// TwinCAT 3 PLC project Untitled1
// ProgramVersion: 3.1.4024.0
// libraries:
//   SPT Base Types, * (Beckhoff Automation LLC)
//   SPT Components, * (Beckhoff Automation LLC)
//   SPT Event Logger, * (Beckhoff Automation LLC)
//   SPT Motion Control, * (Beckhoff Automation LLC)
//   Tc2_EtherCAT, * (Beckhoff Automation GmbH)
//   Tc2_Standard, * (Beckhoff Automation GmbH)
//   Tc2_System, * (Beckhoff Automation GmbH)
//   Tc3_EventLogger, * (Beckhoff Automation GmbH)
//   Tc3_Module, * (Beckhoff Automation GmbH)
//   Tc3_PackML_V2, * (Beckhoff Automation GmbH)
// project tree:
//   DUTs/ E_PMLCustomMode.TcDUT
//   Machine/01_MachineModule/DUTs/ ST_MachineCommand.TcDUT, ST_MachineConfig.TcDUT, ST_MachineRecipe.TcDUT, ST_MachineStatus.TcDUT
//   Machine/01_MachineModule/ I_MachineModule.TcIO, Machine.TcPOU
//   Machine/02_EquipmentModules/01_Infeed/DUTs/ ST_InfeedConfig.TcDUT, ST_InfeedRecipe.TcDUT, ST_InfeedStatus.TcDUT, ST_InfeedCommand.TcDUT
//   Machine/02_EquipmentModules/01_Infeed/ EM_InfeedModule.TcPOU, I_InfeedModule.TcIO
//   Machine/02_EquipmentModules/02_Process/DUTs/ ST_ProcessCommand.TcDUT, ST_ProcessConfig.TcDUT, ST_ProcessRecipe.TcDUT, ST_ProcessStatus.TcDUT
//   Machine/02_EquipmentModules/02_Process/ EM_ProcessModule.TcPOU, I_ProcessModule.TcIO
//   Machine/02_EquipmentModules/03_Outfeed/DUTs/ ST_OutfeedCommand.TcDUT, ST_OutfeedConfig.TcDUT, ST_OutfeedRecipe.TcDUT, ST_OutfeedStatus.TcDUT
//   Machine/02_EquipmentModules/03_Outfeed/ EM_OutfeedModule.TcPOU, I_OutfeedModule.TcIO
//   Machine/03_Components/ FB_Component_StackLight.TcPOU, FB_Component_TwinSAFE_Monitor.TcPOU
//   / PlcTask.TcTTO
//   POUs/ CD_CommonModule.TcCD (not stored), CD_Visitor.TcCD (not stored), MAIN.TcPOU
//   POUs/Common/Component/ CommonComponent.TcPOU, I_CommonComponent.TcIO
//   POUs/Common/Module/ CommonModule.TcPOU, I_CommonModule.TcIO
//   POUs/Common/Module/DUTs/ ST_CommandCommon.TcDUT, ST_ConfigCommon.TcDUT, ST_RecipeCommon.TcDUT, ST_StatusCommon.TcDUT
//   Visitors/ FB_CollectOEE.TcPOU, I_VisitModules.TcIO
// real-time tasks:
//   TASK PlcTask: cycle T#10ms, priority 20, ADS port 350
// motion (NC):
//   TASK NC-Task 1 SAF: cycle T#2ms, priority 4, ADS port 501
//   TASK NC-Task 1 SVB: cycle T#10ms, priority 8, ADS port 511
//   AXIS Infeed (id 1)
//     OtherSettings: AllowMotionCmdToSlave=true
//     encoder EncType=1
//     drive DrvType=5
//       Analog: TorqueSetpointScale=10, ScaleFactorActTorque=0.1
//     controller CtrType=1
//       CtrPara: PriorControlFactor=1
//         Observer: BandWidth=20
//   AXIS Process (id 2)
//     OtherSettings: AllowMotionCmdToSlave=true
//     encoder EncType=1
//     drive DrvType=5
//       Analog: TorqueSetpointScale=10, ScaleFactorActTorque=0.1
//     controller CtrType=1
//       CtrPara: PriorControlFactor=1
//         Observer: BandWidth=20
//   AXIS Outfeed (id 3)
//     OtherSettings: AllowMotionCmdToSlave=true
//     encoder EncType=1
//     drive DrvType=5
//       Analog: TorqueSetpointScale=10, ScaleFactorActTorque=0.1
//     controller CtrType=1
//       CtrPara: PriorControlFactor=1
//         Observer: BandWidth=20
// variable links:
//   Untitled1/Untitled1 Instance <-> NC-Task 1 SAF/Axes/Infeed
//     PlcTask Inputs/MAIN.Machine.Infeed.Axis.BasicAxis._Axis.NcToPlc <-> Outputs/ToPlc
//     PlcTask Outputs/MAIN.Machine.Infeed.Axis.BasicAxis._Axis.PlcToNc <-> Inputs/FromPlc
//   Untitled1/Untitled1 Instance <-> NC-Task 1 SAF/Axes/Outfeed
//     PlcTask Inputs/MAIN.Machine.Outfeed.Axis.BasicAxis._Axis.NcToPlc <-> Outputs/ToPlc
//     PlcTask Outputs/MAIN.Machine.Outfeed.Axis.BasicAxis._Axis.PlcToNc <-> Inputs/FromPlc
//   Untitled1/Untitled1 Instance <-> NC-Task 1 SAF/Axes/Process
//     PlcTask Inputs/MAIN.Machine.Process.Axis.BasicAxis._Axis.NcToPlc <-> Outputs/ToPlc
//     PlcTask Outputs/MAIN.Machine.Process.Axis.BasicAxis._Axis.PlcToNc <-> Inputs/FromPlc

CONFIGURATION Untitled1
    RESOURCE PLC ON TwinCAT3
        TASK PlcTask(INTERVAL := T#10ms, PRIORITY := 20);
        PROGRAM MAIN WITH PlcTask : MAIN;
    END_RESOURCE
END_CONFIGURATION

// ---- DUTs/E_PMLCustomMode.TcDUT
{attribute 'to_string'}
TYPE E_PMLCustomMode : (
		//Reserved
		Production	:= 1,
		Maintenance := 2,
		Manual		:= 3,
		//User-Defined
		Home		   := 4,
		PrePositioning := 5,
		PreHeating	   := 6,
		PreProduction  := 7,
		SingleCycle	   := 8,
		SingleStep	   := 9,
		SetupMode	   := 10,
		CleanInPlace   := 11
	) DINT;
END_TYPE

// ---- Machine/01_MachineModule/DUTs/ST_MachineCommand.TcDUT
TYPE ST_MachineCommand :
	STRUCT
		LightOn : BOOL;
	END_STRUCT
END_TYPE

// ---- Machine/01_MachineModule/DUTs/ST_MachineConfig.TcDUT
TYPE ST_MachineConfig :
	STRUCT
	END_STRUCT
END_TYPE

// ---- Machine/01_MachineModule/DUTs/ST_MachineRecipe.TcDUT
TYPE ST_MachineRecipe :
	STRUCT
	END_STRUCT
END_TYPE

// ---- Machine/01_MachineModule/DUTs/ST_MachineStatus.TcDUT
TYPE ST_MachineStatus :
	STRUCT
	END_STRUCT
END_TYPE

// ---- Machine/02_EquipmentModules/01_Infeed/DUTs/ST_InfeedConfig.TcDUT
TYPE ST_InfeedConfig :
	STRUCT
	END_STRUCT
END_TYPE

// ---- Machine/02_EquipmentModules/01_Infeed/DUTs/ST_InfeedRecipe.TcDUT
TYPE ST_InfeedRecipe :
	STRUCT
	END_STRUCT
END_TYPE

// ---- Machine/02_EquipmentModules/01_Infeed/DUTs/ST_InfeedStatus.TcDUT
TYPE ST_InfeedStatus :
	STRUCT
		ConveyorRunning : BOOL;
	END_STRUCT
END_TYPE

// ---- Machine/02_EquipmentModules/01_Infeed/DUTs/ST_InfeedCommand.TcDUT
TYPE ST_InfeedCommand :
	STRUCT
		StartConveyor : BOOL;
		StopConveyor  : BOOL;
	END_STRUCT
END_TYPE

// ---- Machine/02_EquipmentModules/02_Process/DUTs/ST_ProcessCommand.TcDUT
TYPE ST_ProcessCommand :
	STRUCT
		MoveToAbortPos : BOOL;
	END_STRUCT
END_TYPE

// ---- Machine/02_EquipmentModules/02_Process/DUTs/ST_ProcessConfig.TcDUT
TYPE ST_ProcessConfig :
	STRUCT
	END_STRUCT
END_TYPE

// ---- Machine/02_EquipmentModules/02_Process/DUTs/ST_ProcessRecipe.TcDUT
TYPE ST_ProcessRecipe :
	STRUCT
		RollTime : TIME := T#1S;
	END_STRUCT
END_TYPE

// ---- Machine/02_EquipmentModules/02_Process/DUTs/ST_ProcessStatus.TcDUT
TYPE ST_ProcessStatus :
	STRUCT
		ProductAtReady	: BOOL;
		ProductInPos	: BOOL;
		ProcessComplete : BOOL;
	END_STRUCT
END_TYPE

// ---- Machine/02_EquipmentModules/03_Outfeed/DUTs/ST_OutfeedCommand.TcDUT
TYPE ST_OutfeedCommand :
	STRUCT
		StartConveyor : bool;
		StopConveyor : BOOL;
	END_STRUCT
END_TYPE

// ---- Machine/02_EquipmentModules/03_Outfeed/DUTs/ST_OutfeedConfig.TcDUT
TYPE ST_OutfeedConfig :
	STRUCT
	END_STRUCT
END_TYPE

// ---- Machine/02_EquipmentModules/03_Outfeed/DUTs/ST_OutfeedRecipe.TcDUT
TYPE ST_OutfeedRecipe :
	STRUCT
	END_STRUCT
END_TYPE

// ---- Machine/02_EquipmentModules/03_Outfeed/DUTs/ST_OutfeedStatus.TcDUT
TYPE ST_OutfeedStatus :
	STRUCT
		ProductAtReady	: BOOL;
		ProductRemoved	: BOOL;
		ConveyorRunning : BOOL;
	END_STRUCT
END_TYPE

// ---- POUs/Common/Module/DUTs/ST_CommandCommon.TcDUT
TYPE ST_CommandCommon EXTENDS ST_PackMLBaseModule_Command :
	STRUCT
		Home		   : BOOL;
		Start		   : BOOL;
		Reset		   : BOOL;
		EmergencyStop  : BOOL;
		ControlledStop : BOOL;
	END_STRUCT
END_TYPE

// ---- POUs/Common/Module/DUTs/ST_ConfigCommon.TcDUT
TYPE ST_ConfigCommon :
STRUCT
END_STRUCT
END_TYPE

// ---- POUs/Common/Module/DUTs/ST_RecipeCommon.TcDUT
TYPE ST_RecipeCommon :
STRUCT
END_STRUCT
END_TYPE

// ---- POUs/Common/Module/DUTs/ST_StatusCommon.TcDUT
TYPE ST_StatusCommon EXTENDS ST_PackMLBaseModule_Status :
	STRUCT
		Homed : BOOL;
	END_STRUCT
END_TYPE

// ---- Machine/01_MachineModule/I_MachineModule.TcIO
INTERFACE I_MachineModule

PROPERTY CfgMachine : REFERENCE TO ST_MachineConfig
GET
END_GET
END_PROPERTY

PROPERTY CmdMachine : REFERENCE TO ST_MachineCommand
GET
END_GET
END_PROPERTY

PROPERTY RcpMachine : REFERENCE TO ST_MachineRecipe
GET
END_GET
END_PROPERTY

PROPERTY StsMachine : REFERENCE TO ST_MachineStatus
GET
END_GET
END_PROPERTY

END_INTERFACE

// ---- Machine/02_EquipmentModules/01_Infeed/I_InfeedModule.TcIO
INTERFACE I_InfeedModule

PROPERTY CfgInfeed : REFERENCE TO ST_InfeedConfig
GET
END_GET
END_PROPERTY

PROPERTY CmdInfeed : REFERENCE TO ST_InfeedCommand
GET
END_GET
END_PROPERTY

PROPERTY RcpInfeed : REFERENCE TO ST_InfeedRecipe
GET
END_GET
END_PROPERTY

PROPERTY StsInfeed : REFERENCE TO ST_InfeedStatus
GET
END_GET
END_PROPERTY

END_INTERFACE

// ---- Machine/02_EquipmentModules/02_Process/I_ProcessModule.TcIO
INTERFACE I_ProcessModule

PROPERTY CfgProcess : REFERENCE TO ST_ProcessConfig
GET
END_GET
END_PROPERTY

PROPERTY CmdProcess : REFERENCE TO ST_ProcessCommand
GET
END_GET
END_PROPERTY

PROPERTY RcpProcess : REFERENCE TO ST_ProcessRecipe
GET
END_GET
END_PROPERTY

PROPERTY StsProcess : REFERENCE TO ST_ProcessStatus
GET
END_GET
END_PROPERTY

END_INTERFACE

// ---- Machine/02_EquipmentModules/03_Outfeed/I_OutfeedModule.TcIO
INTERFACE I_OutfeedModule

PROPERTY CfgOutfeed : REFERENCE TO ST_OutfeedConfig
GET
END_GET
END_PROPERTY

PROPERTY CmdOutfeed : REFERENCE TO ST_OutfeedCommand
GET
END_GET
END_PROPERTY

PROPERTY RcpOutfeed : REFERENCE TO ST_OutfeedRecipe
GET
END_GET
END_PROPERTY

PROPERTY StsOutfeed : REFERENCE TO ST_OutfeedStatus
GET
END_GET
END_PROPERTY

END_INTERFACE

// ---- POUs/Common/Component/I_CommonComponent.TcIO
INTERFACE I_CommonComponent EXTENDS I_ComponentBase

END_INTERFACE

// ---- POUs/Common/Module/I_CommonModule.TcIO
INTERFACE I_CommonModule EXTENDS I_PackML_BaseModule

METHOD Accept
VAR_INPUT
	Visitor : I_VisitModules;
END_VAR
END_METHOD

PROPERTY CfgCommon : reference to ST_ConfigCommon
GET
END_GET
END_PROPERTY

PROPERTY CmdCommon : REFERENCE TO ST_CommandCommon
GET
END_GET
END_PROPERTY

PROPERTY RcpCommon : reference to ST_RecipeCommon
GET
END_GET
END_PROPERTY

PROPERTY StsCommon : REFERENCE TO ST_StatusCommon
GET
END_GET
END_PROPERTY

END_INTERFACE

// ---- Visitors/I_VisitModules.TcIO
INTERFACE I_VisitModules

METHOD VisitModule : BOOL
VAR_INPUT
	Module : I_CommonModule;
END_VAR
END_METHOD

END_INTERFACE

// ---- POUs/MAIN.TcPOU
PROGRAM MAIN
VAR
	Machine		   : Machine := (Name := 'Machine');
	Reset		   : BOOL;
	Home		   : BOOL;
	Start		   : BOOL;
	Stop		   : BOOL;
	ControlledStop : BOOL;
	EmergencyStop  : BOOL;
END_VAR

(*
	This sample was built to show a few different ways of implementing the various parts of the SPT Framework.
	While the SPT Framework provides the FB_PackML_BaseModule, this Class focuses on providing the necessities from which to build upon.
	
	This sample uses a CommonModule Class that inheirts from the FB_PackML_BaseModule, and does most of the work for managing the state machine of the system's modules.
		This allows for the code that interacts with the Components of a Module to be the primary focuis of the EM.
 	The CommonModule implements the Command and Status Structures which allows for interaction with a modules state machine. Common commands such as Start, Stop, Reset, and Home 
		are sent through the CmdCommon structure. Common Status of the modules can be read through the StsCommon structure.
	For consistency each Equipment Module also has a Cmd and Sts structure named for the EM; for example, CmdInfeed or StsProcess. 
		These hold the more specific EM commands such as Conveyor Start and Conveyor Stop, and a similar Status structure for Conveyor Running or Cylinder Extended.
		It is important to note that all of these structures have a concrete instance defined within the EM, and a property getter that gets a reference to that concretion. 
		This means that it is possible to read and write to the structure through the getter of the propoerty.
	This overall design allows for the code to Stop, Reset, Enable/Disable; that most all components are going to need, to be placed in the CommonModule. Thereby providing the possibility
		to reduce the code in the EMs to only managing what is unique about the EM. This does require the use of interfaces and the __QUERYINTERFACE method, 
		in order to only send axis command to an axis, but it does allow us to efficiently send commands to all axes within an EM at the same time.
		Additionally, if components built by the user implement a common interface to a structure then these components can all be managed through that interface from the CommonModule.
		
	IMPORTANT NOTE:
	The CommonModule makes extensive use of the variable SequenceState throughout the Acting and Execute methods. 
	Therefore it is reccomend to only use the DescendantSequenceState variable within the EMs.
	
*)
Machine.CyclicLogic();

(*
If Not Homed Abort -> Idle, Change Mode to Home, Idle -> Execute
If Homed Abort -> Idle in Mode Production *)
IF Reset THEN
	Reset					:= FALSE;
	Machine.CmdCommon.Reset := TRUE; //Needs to be ignored if state not valid for reset
END_IF

(*
In Home.Execute start Homing Sequence
After Homing finished, Execute -> Suspended, ModeChange to Production *)
IF Home THEN
	Home				   := FALSE;
	Machine.CmdCommon.Home := TRUE; ////Needs to be ignored if state not valid for Home
END_IF

(*
Production.Idle -> Execute
Production.Suspended -> Execute *)
IF Start THEN
	Start					:= FALSE;
	Machine.CmdCommon.Start := TRUE; //Needs to be ignored if state not valid for start
END_IF

IF ControlledStop THEN
	ControlledStop					 := FALSE;
	Machine.CmdCommon.ControlledStop := TRUE;
	Machine.ChangeState(State := E_PMLCommand.ePMLCommand_Stop);
END_IF

IF EmergencyStop THEN
	EmergencyStop					:= FALSE;
	Machine.CmdCommon.EmergencyStop := TRUE;
	Machine.ChangeState(State := E_PMLCommand.ePMLCommand_Abort);
END_IF

END_PROGRAM

// ---- Machine/01_MachineModule/Machine.TcPOU
FUNCTION_BLOCK Machine EXTENDS CommonModule IMPLEMENTS I_MachineModule
VAR
	//EMs
	Infeed	: EM_InfeedModule  := (Name := 'Infeed');
	Process : EM_ProcessModule := (Name := 'Process');
	Outfeed : EM_OutfeedModule := (Name := 'Outfeed');

	//Components
	StackLight		 : FB_Component_StackLight		 := (Name := 'StackLight');
	TwinSAFE_Monitor : FB_Component_TwinSAFE_Monitor := (Name := 'TwinSAFE_Monitor');

	//
	fbTON_InfeedRun	   : TON;
	fbTON_ProcessDelay : TON;
	fbTON_OutfeedRun   : TON;

	//
	_CmdMachine : ST_MachineCommand;
	_StsMachine : ST_MachineStatus;
	_RcpMachine : ST_MachineRecipe;
	_CfgMachine : ST_MachineConfig;

	//Visitor
	CollectOEE_MM : FB_CollectOEE;
END_VAR

PROPERTY CfgMachine : REFERENCE TO ST_MachineConfig
GET
CfgMachine REF= _CfgMachine;
END_GET
END_PROPERTY

PROPERTY CmdMachine : REFERENCE TO ST_MachineCommand
GET
CmdMachine REF= _CmdMachine;
END_GET
END_PROPERTY

METHOD CreateCustomModes : BOOL
VAR_INPUT
END_VAR
//Production
CustomModes(eMode						   := E_PMLCustomMode.Production,
			sName						   := 'Production',
			bDisableClearing			   := FALSE,
			bDisableStarting			   := FALSE,
			bDisableSuspended			   := FALSE,
			bDisableStopping			   := FALSE,
			bDisableAborting			   := FALSE,
			bDisableHolding				   := FALSE,
			bDisableHeld				   := FALSE,
			bDisableUnholding			   := FALSE,
			bDisableSuspending			   := FALSE,
			bDisableUnsuspending		   := FALSE,
			bDisableResetting			   := FALSE,
			bDisableIdle				   := FALSE,
			bDisableCompleting			   := FALSE,
			bDisableComplete			   := FALSE,
			bEnableUnitModeChangeStopped   := TRUE,
			bEnableUnitModeChangeIdle	   := TRUE,
			bEnableUnitModeChangeSuspended := TRUE,
			bEnableUnitModeChangeExecute   := TRUE,
			bEnableUnitModeChangeAborted   := TRUE,
			bEnableUnitModeChangeHeld	   := TRUE,
			bEnableUnitModeChangeComplete  := TRUE);

//Home
CustomModes(eMode						   := E_PMLCustomMode.Home,
			sName						   := 'Home',
			bDisableClearing			   := FALSE,
			bDisableStarting			   := FALSE,
			bDisableSuspended			   := FALSE,
			bDisableStopping			   := FALSE,
			bDisableAborting			   := FALSE,
			bDisableHolding				   := FALSE,
			bDisableHeld				   := FALSE,
			bDisableUnholding			   := FALSE,
			bDisableSuspending			   := FALSE,
			bDisableUnsuspending		   := FALSE,
			bDisableResetting			   := FALSE,
			bDisableIdle				   := FALSE,
			bDisableCompleting			   := FALSE,
			bDisableComplete			   := FALSE,
			bEnableUnitModeChangeStopped   := TRUE,
			bEnableUnitModeChangeIdle	   := TRUE,
			bEnableUnitModeChangeSuspended := TRUE,
			bEnableUnitModeChangeExecute   := TRUE,
			bEnableUnitModeChangeAborted   := TRUE,
			bEnableUnitModeChangeHeld	   := TRUE,
			bEnableUnitModeChangeComplete  := TRUE);

//Pre-Positioning for resetting between products
CustomModes(eMode						   := E_PMLCustomMode.PrePositioning,
			sName						   := 'Pre-Positioning',
			bDisableClearing			   := FALSE,
			bDisableStarting			   := FALSE,
			bDisableSuspended			   := FALSE,
			bDisableStopping			   := FALSE,
			bDisableAborting			   := FALSE,
			bDisableHolding				   := FALSE,
			bDisableHeld				   := FALSE,
			bDisableUnholding			   := FALSE,
			bDisableSuspending			   := FALSE,
			bDisableUnsuspending		   := FALSE,
			bDisableResetting			   := FALSE,
			bDisableIdle				   := FALSE,
			bDisableCompleting			   := FALSE,
			bDisableComplete			   := FALSE,
			bEnableUnitModeChangeStopped   := TRUE,
			bEnableUnitModeChangeIdle	   := TRUE,
			bEnableUnitModeChangeSuspended := TRUE,
			bEnableUnitModeChangeExecute   := TRUE,
			bEnableUnitModeChangeAborted   := TRUE,
			bEnableUnitModeChangeHeld	   := TRUE,
			bEnableUnitModeChangeComplete  := TRUE);

//Pre-Production for Heaters
CustomModes(eMode						   := E_PMLCustomMode.PreProduction,
			sName						   := 'Pre-Production',
			bDisableClearing			   := FALSE,
			bDisableStarting			   := FALSE,
			bDisableSuspended			   := FALSE,
			bDisableStopping			   := FALSE,
			bDisableAborting			   := FALSE,
			bDisableHolding				   := FALSE,
			bDisableHeld				   := FALSE,
			bDisableUnholding			   := FALSE,
			bDisableSuspending			   := FALSE,
			bDisableUnsuspending		   := FALSE,
			bDisableResetting			   := FALSE,
			bDisableIdle				   := FALSE,
			bDisableCompleting			   := FALSE,
			bDisableComplete			   := FALSE,
			bEnableUnitModeChangeStopped   := TRUE,
			bEnableUnitModeChangeIdle	   := TRUE,
			bEnableUnitModeChangeSuspended := TRUE,
			bEnableUnitModeChangeExecute   := TRUE,
			bEnableUnitModeChangeAborted   := TRUE,
			bEnableUnitModeChangeHeld	   := TRUE,
			bEnableUnitModeChangeComplete  := TRUE);
END_METHOD

METHOD PUBLIC CyclicLogic
IF NOT _InitComplete THEN
	_InitComplete := Initialize();
	RETURN;
END_IF

//Visitor
Accept(Visitor := CollectOEE_MM);
SUPER^.CyclicLogic();
END_METHOD

//! @summary This method contains code which will execute when this PackML module is in the <b>Execute</b> state
METHOD PROTECTED Execute
(*! <description> <b>The base implementation of this method is empty. User must override this method to provide functionality.</b>
<table> 
	<tr>
		<th> Previous State </th>
		<th> Transition In </th>
		<th> Transition Out </th>
		<th> Next State  </th> 
	</tr>
	<tr>
		<td> Starting<b>-or-</b>Unholding <b>-or-</b>Unsuspending</td>
		<td> State Complete<i>(Starting<b>-or-</b>Unholding<b>-or-</b>Unsuspending)</i></td> 
		<td> State Complete<b>-or-</b>Hold Command<b>-or-</b>Suspend Command</td>
		<td> Completing<b>-or-</b>Holding<b>-or-</b>Suspending</td>
	</tr>
</table>
This method is called as required by <c>StateControl()</c>
</description> 

*)
VAR
END_VAR
CASE _CurrentMode OF
	E_PMLCustomMode.Production:
		CASE DescendantSequenceState OF
			0:
				Infeed.CmdInfeed.StartConveyor := TRUE;
				IF Infeed.StsInfeed.ConveyorRunning THEN
					Infeed.CmdInfeed.StartConveyor := FALSE;
					fbTON_InfeedRun(IN := FALSE);
					DescendantSequenceState := DescendantSequenceState + 10;
				END_IF

			10:
				fbTON_InfeedRun(IN := TRUE, PT := T#3S);
				IF fbTON_InfeedRun.Q THEN
					Infeed.CmdInfeed.StopConveyor := TRUE;
					DescendantSequenceState		  := DescendantSequenceState + 10;
				END_IF

			20:
				IF NOT Infeed.StsInfeed.ConveyorRunning THEN
					Infeed.CmdInfeed.StopConveyor	  := FALSE;
					Process.StsProcess.ProductAtReady := TRUE;
					fbTON_ProcessDelay(IN := FALSE);
					DescendantSequenceState := DescendantSequenceState + 10;
				END_IF

			30:
				fbTON_ProcessDelay(IN := TRUE, PT := T#1.5S);
				IF fbTON_ProcessDelay.Q THEN
					Process.StsProcess.ProductAtReady := FALSE;
					Process.StsProcess.ProductInPos	  := TRUE;
					DescendantSequenceState			  := DescendantSequenceState + 10;
				END_IF

			40:
				IF Process.StsProcess.ProcessComplete THEN
					Process.StsProcess.ProcessComplete := FALSE;
					Outfeed.StsOutfeed.ProductAtReady  := TRUE;
					DescendantSequenceState			   := DescendantSequenceState + 10;
				END_IF

			50:
				IF Outfeed.StsOutfeed.ConveyorRunning THEN
					Outfeed.StsOutfeed.ProductAtReady := FALSE;
					fbTON_OutfeedRun(IN := FALSE);
					DescendantSequenceState := DescendantSequenceState + 10;
				END_IF

			60:
				fbTON_OutfeedRun(IN := TRUE, PT := T#3S);
				IF fbTON_OutfeedRun.Q THEN
					Outfeed.StsOutfeed.ProductRemoved := TRUE;
					DescendantSequenceState			  := DescendantSequenceState + 10;
				END_IF

			70:
				IF NOT Outfeed.StsOutfeed.ConveyorRunning THEN
					Outfeed.StsOutfeed.ProductRemoved := FALSE;
					DescendantSequenceState			  := 0;
				END_IF
		END_CASE

	E_PMLCustomMode.Home:
		_StsCommon.Homed := TRUE;
END_CASE

SUPER^.Execute();
END_METHOD

METHOD PROTECTED Initialize : BOOL
VAR
	i: UDINT;
END_VAR
Initialize := FALSE;
CASE DescendantSequenceState OF
	0: //Register Modules
		RegisterSubmodule(Infeed);
		RegisterSubmodule(Process);
		RegisterSubmodule(Outfeed);

		//Register Components
		RegisterComponent(StackLight);

		//I_CommonModule
		ipCommonModules[1] := Infeed;
		ipCommonModules[2] := Process;
		ipCommonModules[3] := Outfeed;

		//I_CommonComponent
		ipComponents[1] := StackLight;

		//Setup Config
		_LogModeChanges			:= FALSE;
		_LogStateChanges		:= FALSE;
		DescendantSequenceState := DescendantSequenceState + 10;

	10: // Configure Custom Modes
		CreateCustomModes();

		// Copy Mode names
		FOR i := 1 TO 10 DO
			ModeNames[i] := F_UnitModeToString(UDINT_TO_DINT(i));
		END_FOR

		DescendantSequenceState := DescendantSequenceState + 10;

	20:
		//Initialize_Recipes();
		DescendantSequenceState := DescendantSequenceState + 10;

	30: // Call the Super 
		IF SUPER^.Initialize() THEN
			DescendantSequenceState := DescendantSequenceState + 10;
		END_IF

	40:
		Initialize := TRUE;
END_CASE
END_METHOD

PROPERTY RcpMachine : REFERENCE TO ST_MachineRecipe
GET
RcpMachine REF= _RcpMachine;
END_GET
END_PROPERTY

PROPERTY StsMachine : reference to ST_MachineStatus
GET
StsMachine REF= _StsMachine;
END_GET
END_PROPERTY

END_FUNCTION_BLOCK

// ---- POUs/Common/Module/CommonModule.TcPOU
FUNCTION_BLOCK CommonModule EXTENDS FB_PackML_BaseModule IMPLEMENTS I_CommonModule
VAR
	//
	ipCommonModules : ARRAY[1..3] OF I_CommonModule;
	ipCommonModule	: I_CommonModule;
	ipBasicAxis		: I_BasicAxis;
	ipProcessModule : I_ProcessModule;

	//
	_CmdCommon : ST_CommandCommon;
	_StsCommon : ST_StatusCommon;
	_CfgCommon : ST_ConfigCommon;
	_RcpCommon : ST_RecipeCommon;

	//Debug Help
	aCurrentState : ARRAY[1..3] OF E_PMLState;



	//Visitor
	CollectOEE_EMs : ARRAY[1..3] OF FB_CollectOEE;
END_VAR

//! @summary This method contains code which will execute when this PackML module is in the <b>Aborted</b> state
METHOD PROTECTED Aborted

(*! <description> <b>The base implementation of this method is empty. User must override this method to provide functionality.</b>
<table> 
	<tr>
		<th> Previous State </th>
		<th> Transition In </th>
		<th> Transition Out </th>
		<th> Next State  </th> 
	</tr>
	<tr>
		<td> Aborting </td>
		<td> State Complete <i>(Aborting)</i></td> 
		<td> Clear Command </td>
		<td> Clearing </td> 
	</tr>
</table>
This method is called as required by <c>StateControl()</c>
</description> 

*)
IF _CmdCommon.Reset THEN
	//_Cmd.Reset := FALSE;//If used, then the reset button will need to be pressed twice after Abort
	_CmdCommon.EmergencyStop := FALSE;
	ChangeState(State := E_PMLCommand.ePMLCommand_Clear);
END_IF
END_METHOD

//! @summary This method contains code which will execute when this PackML module is in the <b>Aborting</b> state
METHOD PROTECTED Aborting
VAR
	i				: UDINT;
	SubModulesReady : BOOL := TRUE;
	AllAxesDone		: BOOL;
END_VAR

(*! <description> <b>Note:</b> The <i>Abort</i> command should be associated with the fault handing routine of a module. It should not be directly commanded from any user inteface. 

<table> 
	<tr>
		<th> Previous State </th>
		<th> Transition In </th>
		<th> Transition Out </th>
		<th> Next State  </th> 
	</tr>
	<tr>
		<td> <b>ANY</b> </td>
		<td> Abort Command </td> 
		<td> State Complete </td>
		<td> Aborted </td> 
	</tr>
</table>

This method is called as required by <c>StateControl()</c>
</description> 

*)
CASE SequenceState OF
	0:
		NoStateTasksToComplete := FALSE;
		SequenceState		   := SequenceState + 10;

	10:
		//Stop all motion axes
		FOR i := 1 TO NumberOfComponents DO
			IF __QUERYINTERFACE(ipComponents[i], ipBasicAxis) THEN
				IF NOT ipBasicAxis.Stopped THEN
					ipBasicAxis.Stop();
				END_IF
			END_IF
		END_FOR

		SequenceState := SequenceState + 10;

	20:
		//Wait for all motion axes to be stopped
		AllAxesDone := TRUE;
		FOR i := 1 TO NumberOfComponents DO
			IF __QUERYINTERFACE(ipComponents[i], ipBasicAxis) THEN
				IF NOT ipBasicAxis.Stopped THEN
					AllAxesDone := FALSE;
				END_IF
			END_IF
		END_FOR

		IF AllAxesDone THEN
			SequenceState := SequenceState + 10;
		END_IF

	30:
		//Disable all motion axes
		FOR i := 1 TO NumberOfComponents DO
			IF __QUERYINTERFACE(ipComponents[i], ipBasicAxis) THEN
				IF ipBasicAxis.Enabled THEN
					ipBasicAxis.Disable();
				END_IF
			END_IF
		END_FOR

		SequenceState := SequenceState + 10;

	40:
		//Wait for all motion axes to be Disabled
		AllAxesDone := TRUE;
		FOR i := 1 TO NumberOfComponents DO
			IF __QUERYINTERFACE(ipComponents[i], ipBasicAxis) THEN
				IF ipBasicAxis.Enabled THEN
					AllAxesDone := FALSE;
				END_IF
			END_IF
		END_FOR

		IF AllAxesDone THEN
			SequenceState := SequenceState + 10;
		END_IF

	50: //ipCommonModules
		FOR i := 1 TO NumberOfComponents DO
			IF __QUERYINTERFACE(ipCommonModules[i], ipProcessModule) THEN
				ipProcessModule.CmdProcess.MoveToAbortPos := TRUE;
			END_IF
		END_FOR

		SequenceState := SequenceState + 10;

	60:
		StateTasksComplete := true;
END_CASE

SUPER^.Aborting();
END_METHOD

METHOD Accept
VAR_INPUT
	Visitor : I_VisitModules;
END_VAR
Visitor.VisitModule(THIS^);
END_METHOD

PROPERTY CfgCommon : reference to ST_ConfigCommon
GET
CfgCommon REF= _CfgCommon;
END_GET
END_PROPERTY

//! @summary This method contains code which will execute when this PackML module is in the <b>Clearing</b> state
METHOD PROTECTED Clearing
VAR
	i					 : UDINT;
	SubModulesReady		 : BOOL := TRUE;
	AllAxesEnabled : BOOL;
	AllComponentsDone	 : BOOL;
END_VAR

(*! <description> <b>Note:</b> The <i>Clear</i> command can also be thought of as a <i>fault reset</i> depite the ambiguity in the naming of the <i>Reset</i> state. 
<table> 
	<tr>
		<th> Previous State </th>
		<th> Transition In </th>
		<th> Transition Out </th>
		<th> Next State  </th> 
	</tr>
	<tr>
		<td> Aborted </td>
		<td> Clear Command </td> 
		<td> State Complete </td>
		<td> Stopped </td> 
	</tr>
</table>
This method is called as required by <c>StateControl()</c>
</description> 

*)
CASE _CurrentMode OF
	E_PMLCustomMode.Production, E_PMLCustomMode.Home:
		CASE SequenceState OF
			0:
				NoStateTasksToComplete := FALSE;
				SequenceState		   := SequenceState + 10;

			10:
				//Reset and ENable All Axes
				AllAxesEnabled := TRUE;
				FOR i := 1 TO NumberOfComponents DO
					IF __QUERYINTERFACE(ipComponents[i], ipBasicAxis) THEN
						IF NOT ipBasicAxis.Error THEN
							ipBasicAxis.Enable();
						ELSE
							ipBasicAxis.Reset();
							AllAxesEnabled := FALSE;
						END_IF
					END_IF
				END_FOR

				IF AllAxesEnabled THEN
					SequenceState := SequenceState + 10;
				END_IF

			20:
				StateTasksComplete := TRUE;
		END_CASE
END_CASE

SUPER^.Clearing();
END_METHOD

PROPERTY CmdCommon : REFERENCE TO ST_CommandCommon
GET
CmdCommon REF= _CmdCommon;
END_GET
END_PROPERTY

//! @summary This method contains code which will execute when this PackML module is in the <b>Complete</b> state
METHOD PROTECTED Complete

(*! <description> <b>The base implementation of this method is empty. User must override this method to provide functionality.</b>
<table> 
	<tr>
		<th> Previous State </th>
		<th> Transition In </th>
		<th> Transition Out </th>
		<th> Next State  </th> 
	</tr>
	<tr>
		<td> Completing </td>
		<td> State Complete <i>(Completing)</i></td> 
		<td> Reset Command </td>
		<td> Resetting </td> 
	</tr>
</table>
This method is called as required by <c>StateControl()</c>
</description> 

*)
END_METHOD

//! @summary This method monitors <b>components</b> within this PackML module and initiates fault responses as required
METHOD PROTECTED ComponentMonitor : BOOL
VAR
	AlarmResponses : ARRAY[0..4] OF E_AlarmResponse; //Temporary response array
	i			   : UDINT;
END_VAR

//! @description This method is called cyclically by <c>CyclicLogic()</c>
SUPER^.ComponentMonitor();
IF NumberOfComponents <> 0 THEN (* Update alarm severity from components *)
	FOR i := 1 TO NumberOfComponents DO
		IF ipComponents[i].CurrentAlarmSeverity > _CurrentAlarmSeverity THEN
			_CurrentAlarmSeverity := ipComponents[i].CurrentAlarmSeverity;
		END_IF
	END_FOR
END_IF
END_METHOD

METHOD PUBLIC CyclicLogic
VAR
	i : UDINT;
END_VAR
IF NOT _InitComplete THEN
	_InitComplete := Initialize();
	RETURN;
END_IF

//Debug Help
FOR i := 1 TO 3 DO
	IF ipSubModules[i] <> 0 THEN
		aCurrentState[i] := ipSubModules[i].CurrentState;
	END_IF
END_FOR

_StsCommon.Mode	 := _CurrentMode;
_StsCommon.State := _CurrentState;
_CmdCommon.Mode	 := _CommandedMode;
_CmdCommon.State := _CommandedState;

//Visitor
FOR i := 1 TO 3 DO
	IF ipCommonModules[i] <> 0 THEN
		ipCommonModules[i].Accept(Visitor := CollectOEE_EMs[i]);
	END_IF
END_FOR


SUPER^.CyclicLogic();
END_METHOD

//! @summary This method contains code which will execute when this PackML module is in the <b>Execute</b> state
METHOD PROTECTED Execute

(*! <description> <b>The base implementation of this method is empty. User must override this method to provide functionality.</b>
<table> 
	<tr>
		<th> Previous State </th>
		<th> Transition In </th>
		<th> Transition Out </th>
		<th> Next State  </th> 
	</tr>
	<tr>
		<td> Starting<b>-or-</b>Unholding <b>-or-</b>Unsuspending</td>
		<td> State Complete<i>(Starting<b>-or-</b>Unholding<b>-or-</b>Unsuspending)</i></td> 
		<td> State Complete<b>-or-</b>Hold Command<b>-or-</b>Suspend Command</td>
		<td> Completing<b>-or-</b>Holding<b>-or-</b>Suspending</td>
	</tr>
</table>
This method is called as required by <c>StateControl()</c>
</description> 

*)
VAR
	allModulesHomed: BOOL;
	i: UDINT;
END_VAR
CASE _CurrentMode OF
	E_PMLCustomMode.Home:
		CASE SequenceState OF
			0:
				IF _CmdCommon.Home THEN
					FOR i := 1 TO SPT_BaseTypes.Parameters_PackML_Base.MAX_NO_OF_SUBMODULES DO
						IF ipCommonModules[i] <> 0 THEN
							ipCommonModules[i].CmdCommon.Home := TRUE;
						END_IF
					END_FOR

					SequenceState := SequenceState + 10;
				END_IF

			10:
				//Monitor all SubModules, when they have completed Homing, Change State to Suspend
				allModulesHomed := TRUE;
				FOR i := 1 TO SPT_BaseTypes.Parameters_PackML_Base.MAX_NO_OF_SUBMODULES DO
					IF ipCommonModules[i] <> 0 THEN
						IF ipCommonModules[i].StsCommon.Homed = FALSE THEN
							allModulesHomed := FALSE;
							EXIT;
						END_IF
					END_IF
				END_FOR

				IF allModulesHomed AND _StsCommon.Homed THEN
					ChangeState(State := ePMLCommand_Suspend);
				END_IF
		END_CASE
END_CASE
END_METHOD

METHOD PROTECTED Idle
VAR
	ChamgeMode		: INT;
	i				: UDINT;
	allModulesHomed : BOOL;
END_VAR
FOR i := 1 TO SPT_BaseTypes.Parameters_PackML_Base.MAX_NO_OF_SUBMODULES DO
	IF ipCommonModules[i] <> 0 THEN
		IF ipCommonModules[i].StsCommon.Homed = FALSE THEN
			_StsCommon.Homed := FALSE;
			EXIT;
		END_IF
	END_IF
END_FOR

IF NOT _StsCommon.Homed THEN
	ChangeMode(Mode := E_PMLCustomMode.Home);
END_IF

CASE _CurrentMode OF
	E_PMLProtectedUnitMode.ePMLProtUnitMode_Production:
		CASE SequenceState OF
			0:
				IF _StsCommon.Homed THEN
					SequenceState := SequenceState + 10;
				END_IF

			10:
				IF _CmdCommon.Start THEN
					_CmdCommon.Start := FALSE;
					ChangeState(State := ePMLCommand_Start);
				END_IF
		END_CASE

	E_PMLCustomMode.Home:
		IF _CmdCommon.Home THEN
			_CmdCommon.Home := FALSE;
			FOR i := 1 TO SPT_BaseTypes.Parameters_PackML_Base.MAX_NO_OF_SUBMODULES DO
				IF ipCommonModules[i] <> 0 THEN
					ipCommonModules[i].CmdCommon.Home := TRUE;
				END_IF
			END_FOR
		END_IF

		ChangeState(State := ePMLCommand_Start);
END_CASE
END_METHOD

METHOD PROTECTED Initialize : BOOL
VAR
	i: UDINT;
END_VAR
Initialize := SUPER^.Initialize();
END_METHOD

PROPERTY RcpCommon : reference to ST_RecipeCommon
GET
RcpCommon REF= _RcpCommon;
END_GET
END_PROPERTY

//! @summary This method contains code which will execute when this PackML module is in the <b>Resetting</b> state
METHOD PROTECTED Resetting
VAR
	i				: UDINT;
	SubModulesReady : BOOL := TRUE;
	AllAxesEnabled: BOOL;
END_VAR

(*! <description> <b>Note:</b> The <i>Reset</i> command can also be thought of as an <i>enable</i> depite the ambiguity in the naming of the <i>Clearing</i> state.
<table> 
	<tr>
		<th> Previous State </th>
		<th> Transition In </th>
		<th> Transition Out </th>
		<th> Next State  </th> 
	</tr>
	<tr>
		<td> Stopped<b>-or-</b>Completed </td>
		<td> Reset Command </td> 
		<td> State Complete </td>
		<td> Idle </td> 
	</tr>
</table>
This method is called as required by <c>StateControl()</c>
</description> 

*)
CASE _CurrentMode OF
	E_PMLCustomMode.Production, E_PMLCustomMode.Home:
		CASE SequenceState OF
			0:
				NoStateTasksToComplete := FALSE;
				SequenceState		   := SequenceState + 10;

			10:
				//Reset and ENable All Axes
				AllAxesEnabled := TRUE;
				FOR i := 1 TO NumberOfComponents DO
					IF __QUERYINTERFACE(ipComponents[i], ipBasicAxis) THEN
						IF NOT ipBasicAxis.Error THEN
							ipBasicAxis.Enable();
						ELSE
							ipBasicAxis.Reset();
							AllAxesEnabled := FALSE;
						END_IF
					END_IF
				END_FOR

				IF AllAxesEnabled THEN
					SequenceState := SequenceState + 10;
				END_IF

			20:
				StateTasksComplete := TRUE;
		END_CASE
END_CASE

SUPER^.Resetting();
END_METHOD

//! @summary This method contains code which will execute when this PackML module is in the <b>Starting</b> state
METHOD PROTECTED Starting
VAR
	i				: UDINT;
	SubModulesReady : BOOL := TRUE;
END_VAR

(*! <description><b></b><table> 
	<tr>
		<th> Previous State </th>
		<th> Transition In </th>
		<th> Transition Out </th>
		<th> Next State  </th> 
	</tr>
	<tr>
		<td> Idle </td>
		<td> Start Command </td> 
		<td> State Complete </td>
		<td> Execute </td> 
	</tr>
</table>
This method is called as required by <c>StateControl()</c>
</description> 

*)
SUPER^.Starting();
END_METHOD

//! @summary This method contains code which will execute when this PackML module is in the <b>Stopped</b> state
METHOD PROTECTED Stopped

(*! <description> <b>The base implementation of this method is empty. User must override this method to provide functionality.</b>
<table> 
	<tr>
		<th> Previous State </th>
		<th> Transition In </th>
		<th> Transition Out </th>
		<th> Next State  </th> 
	</tr>
	<tr>
		<td> Stopping<b>-or-</b>Clearing </td>
		<td> State Complete <i>(Stopping<b>-or-</b>Clearing)</i></td> 
		<td> Reset Command </td>
		<td> Resetting </td> 
	</tr>
</table>
This method is called as required by <c>StateControl()</c>
</description> 

*)
IF _CmdCommon.Reset THEN
	_CmdCommon.Reset		  := FALSE;
	_CmdCommon.ControlledStop := FALSE;
	ChangeState(State := E_PMLCommand.ePMLCommand_Reset);
END_IF
END_METHOD

//! @summary This method contains code which will execute when this PackML module is in the <b>Stopping</b> state
METHOD PROTECTED Stopping
VAR
	i				  : UDINT;
	SubModulesReady	  : BOOL := TRUE;
	AllComponentsDone : BOOL;
END_VAR

(*! <description><b></b><table> 
	<tr>
		<th> Previous State </th>
		<th> Transition In </th>
		<th> Transition Out </th>
		<th> Next State  </th> 
	</tr>
	<tr>
		<td> <b>ANY<i>except</i></b>Stopped<b>-or-</b>Clearing<b>-or-</b>Aborted<b>-or-</b>Aborting</td>
		<td> Stop Command </td> 
		<td> State Complete </td>
		<td> Stopped </td> 
	</tr>
</table>
This method is called as required by <c>StateControl()</c>
</description> 

*)
CASE _CurrentMode OF
	E_PMLCustomMode.Production, E_PMLCustomMode.Home:
		CASE SequenceState OF
			0:
				NoStateTasksToComplete := FALSE;
				SequenceState		   := SequenceState + 10;

			10:
				//Stop all motion axes
				FOR i := 1 TO NumberOfComponents DO
					IF __QUERYINTERFACE(ipComponents[i], ipBasicAxis) THEN
						IF NOT ipBasicAxis.Stopped THEN
							ipBasicAxis.Stop();
						END_IF
					END_IF
				END_FOR

				SequenceState := SequenceState + 10;

			20:
				//Wait for all motion axes to be stopped
				AllComponentsDone := TRUE;
				FOR i := 1 TO NumberOfComponents DO
					IF __QUERYINTERFACE(ipComponents[i], ipBasicAxis) THEN
						IF NOT ipBasicAxis.Stopped THEN
							AllComponentsDone := FALSE;
						END_IF
					END_IF
				END_FOR

				IF AllComponentsDone THEN
					SequenceState := SequenceState + 10;
				END_IF

			30:
				StateTasksComplete := TRUE;
		END_CASE
END_CASE

SUPER^.Stopping();
END_METHOD

PROPERTY StsCommon : REFERENCE TO ST_StatusCommon
GET
StsCommon REF= _StsCommon;
END_GET
END_PROPERTY

//! @summary This method monitors <b>submodules</b> within this PackML module and initiates fault responses as required
METHOD PROTECTED SubModuleMonitor : BOOL
VAR
	AlarmResponses : ARRAY[0..4] OF E_AlarmResponse; //Temporary response array	
	i			   : UDINT;
END_VAR

//! @description This method is called cyclically by <c>CyclicLogic()</c>
SUPER^.SubModuleMonitor();
IF NumberOfSubModules <> 0 THEN (* Update alarm severity from Submodules *)
	FOR i := 1 TO NumberOfSubModules DO
		IF ipSubModules[i].CurrentAlarmSeverity > _CurrentAlarmSeverity THEN
			_CurrentAlarmSeverity := ipSubModules[i].CurrentAlarmSeverity;
		END_IF
	END_FOR
END_IF
END_METHOD

//! @summary This method contains code which will execute when this PackML module is in the <b>Suspended</b> state
METHOD PROTECTED Suspended

(*! <description> <b>The base implementation of this method is empty. User must override this method to provide functionality.</b>
<table> 
	<tr>
		<th> Previous State </th>
		<th> Transition In </th>
		<th> Transition Out </th>
		<th> Next State  </th> 
	</tr>
	<tr>
		<td> Suspending </td>
		<td> State Complete <i>(Suspending)</i></td> 
		<td> Unsuspend Command </td>
		<td> Unsuspending </td> 
	</tr>
</table>
This method is called as required by <c>StateControl()</c>
</description> 

*)
CASE CurrentMode OF
	E_PMLCustomMode.Production:
		IF _CmdCommon.Start THEN
			_CmdCommon.Start := FALSE;
			ChangeState(State := E_PMLCommand.ePMLCommand_Unsuspend);
		END_IF

	E_PMLCustomMode.Home:
		IF _StsCommon.Homed THEN
			ChangeMode(Mode := E_PMLCustomMode.Production);
		END_IF
END_CASE
END_METHOD

//! @summary This method contains code which will execute when this PackML module is in the <b>Suspending</b> state
METHOD PROTECTED Suspending
VAR
	i				: UDINT;
	SubModulesReady : BOOL := TRUE;
END_VAR

(*! <description><b>Note:</b> The <i>Suspend</i> command is intended to be initiated by automatic detection of upstream/downstream jams, etc. It is meant to be distinct from a <i>Hold</i> in that <i>Hold</i> should be commanded by an operator.  Both <i>Hold</i>and<i>Suspend</i> result in a <i>paused</i> state which should allow resumption of the <b>Execute</b> state. 
<table> 
	<tr>
		<th> Previous State </th>
		<th> Transition In </th>
		<th> Transition Out </th>
		<th> Next State  </th> 
	</tr>
	<tr>
		<td> Execute </td>
		<td> Suspend Command </td> 
		<td> State Complete </td>
		<td> Suspended </td> 
	</tr>
</table>
This method is called as required by <c>StateControl()</c>
</description> 

*)
SUPER^.Suspending();
END_METHOD

//! @summary This method contains code which will execute when this PackML module is in the <b>Unsuspending</b> state
METHOD PROTECTED Unsuspending
VAR
	i				: UDINT;
	SubModulesReady : BOOL := TRUE;
END_VAR

(*! <description><b></b><table> 
	<tr>
		<th> Previous State </th>
		<th> Transition In </th>
		<th> Transition Out </th>
		<th> Next State  </th> 
	</tr>
	<tr>
		<td> Suspended </td>
		<td> Unsuspend Command </td> 
		<td> State Complete </td>
		<td> Execute </td> 
	</tr>
</table>
This method is called as required by <c>StateControl()</c>
</description> 

*)
SUPER^.Unsuspending();
END_METHOD

END_FUNCTION_BLOCK

// ---- Visitors/FB_CollectOEE.TcPOU
FUNCTION_BLOCK FB_CollectOEE IMPLEMENTS I_VisitModules
VAR
    _PackTags : ST_PackMLv30Ext;
END_VAR

METHOD UpdateModeTimers
VAR
	currentTime : T_DCTIME64;
END_VAR

VAR_INST
	lastTime	 : T_DCTIME64 := F_GetActualDcTime64();
	lastState	 : DINT;
	lastMode	 : DINT;
	timeDiff	 : LREAL;
	timeToUpdate : LREAL;
END_VAR
IF _PackTags.Status.StateCurrent <> lastState THEN
    MEMSET(ADR(_PackTags.Admin.StateCurrentTime), 0, SIZEOF(_PackTags.Admin.StateCurrentTime));
    lastState := _PackTags.Status.StateCurrent;
END_IF

IF _PackTags.Status.UnitModeCurrent <> lastMode THEN
    MEMSET(ADR(_PackTags.Admin.ModeCurrentTime), 0, SIZEOF(_PackTags.Admin.ModeCurrentTime));
    lastMode := _PackTags.Status.UnitModeCurrent;
END_IF

currentTime := F_GetActualDcTime64();
IF lastTime <> 0 THEN
	//timeToUpdate := ULINT_TO_LREAL(currentTime - lastTime)/1_000_000;
    timeToUpdate := ULINT_TO_LREAL(currentTime - lastTime) / 1_000_000_000.0;
END_IF

// only seconds get added to the cumulative timers 
IF timeToUpdate > 1 THEN
    _PackTags.Admin.ModeCummulativeTime[_PackTags.Status.UnitModeCurrent] := _PackTags.Admin.ModeCummulativeTime[_PackTags.Status.UnitModeCurrent] + LREAL_TO_DINT(timeToUpdate);
    _PackTags.Admin.ModeCurrentTime[_PackTags.Status.UnitModeCurrent]     := _PackTags.Admin.ModeCurrentTime[_PackTags.Status.UnitModeCurrent] + LREAL_TO_DINT(timeToUpdate);
    _PackTags.Admin.StateCummulativeTime[_PackTags.Status.UnitModeCurrent, _PackTags.Status.StateCurrent]
        := _PackTags.Admin.StateCummulativeTime[_PackTags.Status.UnitModeCurrent, _PackTags.Status.StateCurrent] + LREAL_TO_DINT(timeToUpdate);

    _PackTags.Admin.StateCurrentTime[_PackTags.Status.UnitModeCurrent, _PackTags.Status.StateCurrent] :=
        _PackTags.Admin.StateCurrentTime[_PackTags.Status.UnitModeCurrent, _PackTags.Status.StateCurrent] + LREAL_TO_DINT(timeToUpdate);

    lastTime := currentTime;
END_IF
END_METHOD

METHOD VisitModule : BOOL
VAR_INPUT
	Module	: I_CommonModule;
END_VAR
_PackTags.Status.StateCurrent	 := Module.CurrentState;
_PackTags.Status.UnitModeCurrent := Module.CurrentMode;
UpdateModeTimers();
END_METHOD

END_FUNCTION_BLOCK

// ---- Machine/02_EquipmentModules/01_Infeed/EM_InfeedModule.TcPOU
FUNCTION_BLOCK EM_InfeedModule EXTENDS CommonModule IMPLEMENTS I_InfeedModule
VAR
	//Components
	Axis		: FB_Component_BasicAxis;
	

	//
	_CmdInfeed : ST_InfeedCommand;
	_StsInfeed : ST_InfeedStatus;
	_CfgInfeed : ST_InfeedConfig;
	_RcpInfeed : ST_InfeedRecipe;

	//Test Vars
	Homed : BOOL;
END_VAR

PROPERTY CfgInfeed : REFERENCE TO ST_InfeedConfig
GET
CfgInfeed REF= _CfgInfeed;
END_GET
END_PROPERTY

PROPERTY CmdInfeed : REFERENCE TO ST_InfeedCommand
GET
CmdInfeed REF= _CmdInfeed;
END_GET
END_PROPERTY

METHOD PUBLIC CyclicLogic
IF NOT _InitComplete THEN
	_InitComplete := Initialize();
	RETURN;
END_IF

SUPER^.CyclicLogic();
END_METHOD

METHOD PROTECTED Execute
VAR
	i				  : UDINT;
	AllComponentsDone : BOOL;
END_VAR
CASE _CurrentMode OF
	E_PMLCustomMode.Production:
		CASE DescendantSequenceState OF
			0:
				IF _CmdInfeed.StartConveyor THEN
					_CmdInfeed.StartConveyor := FALSE;
					DescendantSequenceState	 := DescendantSequenceState + 10;
				END_IF

			10:
				IF Axis.MoveVelocity(10.0, 0) THEN
					DescendantSequenceState := DescendantSequenceState + 10;
				END_IF

			20:
				IF Axis.Axis.Status.Moving THEN
					_StsInfeed.ConveyorRunning := TRUE;
				END_IF

				IF _CmdInfeed.StopConveyor THEN
					_CmdInfeed.StopConveyor := FALSE;
					Axis.Stop();
					DescendantSequenceState := DescendantSequenceState + 10;
				END_IF

			30:
				IF Axis.Axis.Status.NotMoving THEN
					_StsInfeed.ConveyorRunning := FALSE;
					DescendantSequenceState	   := 0;
				END_IF
		END_CASE

	E_PMLCustomMode.Home:
		CASE DescendantSequenceState OF
			0:
				IF _CmdCommon.Home AND NOT _StsCommon.Homed THEN
					_CmdCommon.Home := FALSE;
					Axis.Home();
					DescendantSequenceState := DescendantSequenceState + 10;
				END_IF

			10:
				IF Axis.Axis.Status.Homed THEN
					_StsCommon.Homed := TRUE;
				END_IF
		END_CASE
END_CASE

SUPER^.Execute();
END_METHOD

METHOD PROTECTED Initialize : BOOL
VAR
	i: UDINT;
END_VAR
Initialize := FALSE;
CASE DescendantSequenceState OF
	0: //Register Modules

		//Register Components
		RegisterComponent(Axis);

		//I_CommonModuleBase

		//I_CommonComponent
		ipComponents[1] := Axis;

		//Setup Config
		_LogModeChanges			:= FALSE;
		_LogStateChanges		:= FALSE;
		DescendantSequenceState := DescendantSequenceState + 10;

	10:
		// Copy Mode names
		FOR i := 1 TO 10 DO
			ModeNames[i] := F_UnitModeToString(UDINT_TO_DINT(i));
		END_FOR

		DescendantSequenceState := DescendantSequenceState + 10;

	20:
		//Initialize_Recipes();
		DescendantSequenceState := DescendantSequenceState + 10;

	30: // Call the Super 
		IF SUPER^.Initialize() THEN
			DescendantSequenceState := DescendantSequenceState + 10;
		END_IF

	40:
		Initialize := TRUE;
END_CASE
END_METHOD

PROPERTY RcpInfeed : REFERENCE TO ST_InfeedRecipe
GET
RcpInfeed REF= _RcpInfeed;
END_GET
END_PROPERTY

PROPERTY StsInfeed : REFERENCE TO ST_InfeedStatus
GET
StsInfeed REF= _StsInfeed;
END_GET
END_PROPERTY

END_FUNCTION_BLOCK

// ---- Machine/02_EquipmentModules/02_Process/EM_ProcessModule.TcPOU
FUNCTION_BLOCK EM_ProcessModule EXTENDS CommonModule IMPLEMENTS I_ProcessModule
VAR
	//Components
	Axis		: FB_Component_BasicAxis;
	Cylinder	: FB_DoubleSolenoidFeedback;
	fbTON_Press : Ton;

	//
	_CmdProcess : ST_ProcessCommand;
	_StsProcess : ST_ProcessStatus;
	_CfgProcess : ST_ProcessConfig;
	_RcpProcess : ST_ProcessRecipe;

	//Test Vars
	Homed : BOOL;
END_VAR

//! @summary This method contains code which will execute when this PackML module is in the <b>Aborting</b> state
METHOD PROTECTED Aborting
VAR
	i				: UDINT;
	SubModulesReady : BOOL := TRUE;
	AllAxesDone		: BOOL;
END_VAR

(*! <description> <b>Note:</b> The <i>Abort</i> command should be associated with the fault handing routine of a module. It should not be directly commanded from any user inteface. 

<table> 
	<tr>
		<th> Previous State </th>
		<th> Transition In </th>
		<th> Transition Out </th>
		<th> Next State  </th> 
	</tr>
	<tr>
		<td> <b>ANY</b> </td>
		<td> Abort Command </td> 
		<td> State Complete </td>
		<td> Aborted </td> 
	</tr>
</table>

This method is called as required by <c>StateControl()</c>
</description> 

*)
CASE DescendantSequenceState OF
	0:
		NoStateTasksToComplete	:= FALSE;
		DescendantSequenceState := DescendantSequenceState + 10;

	10:
		IF _CmdProcess.MoveToAbortPos THEN
			Cylinder.Retract();
		END_IF

		IF Cylinder.Retracted THEN
			DescendantSequenceState := DescendantSequenceState + 10;
		END_IF

	20:
		StateTasksComplete := TRUE;
END_CASE

SUPER^.Aborting();
END_METHOD

PROPERTY CfgProcess : REFERENCE TO ST_ProcessConfig
GET
CfgProcess REF= _CfgProcess;
END_GET
END_PROPERTY

PROPERTY CmdProcess : REFERENCE TO ST_ProcessCommand
GET
CmdProcess REF= _CmdProcess;
END_GET
END_PROPERTY

METHOD PUBLIC CyclicLogic
IF NOT _InitComplete THEN
	_InitComplete := Initialize();
	RETURN;
END_IF

SUPER^.CyclicLogic();
END_METHOD

//! @summary This method contains code which will execute when this PackML module is in the <b>Execute</b> state
METHOD PROTECTED Execute
(*! <description> <b>The base implementation of this method is empty. User must override this method to provide functionality.</b>
<table> 
	<tr>
		<th> Previous State </th>
		<th> Transition In </th>
		<th> Transition Out </th>
		<th> Next State  </th> 
	</tr>
	<tr>
		<td> Starting<b>-or-</b>Unholding <b>-or-</b>Unsuspending</td>
		<td> State Complete<i>(Starting<b>-or-</b>Unholding<b>-or-</b>Unsuspending)</i></td> 
		<td> State Complete<b>-or-</b>Hold Command<b>-or-</b>Suspend Command</td>
		<td> Completing<b>-or-</b>Holding<b>-or-</b>Suspending</td>
	</tr>
</table>
This method is called as required by <c>StateControl()</c>
</description> 

*)
VAR

END_VAR
CASE _CurrentMode OF
	E_PMLCustomMode.Production:
		CASE DescendantSequenceState OF
			0:
				IF _StsProcess.ProductAtReady THEN
					DescendantSequenceState := DescendantSequenceState + 10;
				END_IF

			10:
				IF Axis.MoveVelocity(10.0, 0) THEN
					DescendantSequenceState := DescendantSequenceState + 10;
				END_IF

			20:
				IF _StsProcess.ProductInPos THEN
					Cylinder.Extend();
					fbTON_Press(IN := FALSE);
					DescendantSequenceState := DescendantSequenceState + 10;
				END_IF

			30:
				IF Cylinder.Extended THEN
					fbTON_Press(IN := TRUE, PT := _RcpProcess.RollTime);
				END_IF

				IF fbTON_Press.q THEN
					Cylinder.Retract();
					DescendantSequenceState := DescendantSequenceState + 10;
				END_IF

			40:
				IF Cylinder.Retracted THEN
					Axis.Stop();
					DescendantSequenceState := DescendantSequenceState + 10;
				END_IF

			50:
				IF Axis.Stopped THEN
					_StsProcess.ProcessComplete := TRUE;
					DescendantSequenceState		:= 0;
				END_IF
		END_CASE

	E_PMLCustomMode.Home:
		CASE DescendantSequenceState OF
			0:
				IF _CmdCommon.Home THEN
					Cylinder.Retract();
				END_IF

				IF Cylinder.Retracted THEN
					DescendantSequenceState := DescendantSequenceState + 10;
				END_IF

			10:
				IF _CmdCommon.Home AND NOT _StsCommon.Homed THEN
					_CmdCommon.Home := FALSE;
					Axis.Home();
					DescendantSequenceState := DescendantSequenceState + 10;
				END_IF

			20:
				IF Axis.Axis.Status.Homed THEN
					_StsCommon.Homed := TRUE;
				END_IF
		END_CASE
END_CASE

SUPER^.Execute();
END_METHOD

METHOD PROTECTED Initialize : BOOL
VAR
	i: UDINT;
END_VAR
Initialize := FALSE;
CASE DescendantSequenceState OF
	0: //Register Modules

		//Register Components
		RegisterComponent(Axis);
		RegisterComponent(Cylinder);

		//I_CommonModuleBase

		//I_CommonComponent
		ipComponents[1] := Axis;
		ipComponents[2] := Cylinder;

		//Setup Config
		_LogModeChanges			:= FALSE;
		_LogStateChanges		:= FALSE;
		DescendantSequenceState := DescendantSequenceState + 10;

	10:
		// Copy Mode names
		FOR i := 1 TO 10 DO
			ModeNames[i] := F_UnitModeToString(UDINT_TO_DINT(i));
		END_FOR

		DescendantSequenceState := DescendantSequenceState + 10;

	20:
		//Initialize_Recipes();
		Cylinder.InSimulation	:= TRUE;
		DescendantSequenceState := DescendantSequenceState + 10;

	30: // Call the Super 
		IF SUPER^.Initialize() THEN
			DescendantSequenceState := DescendantSequenceState + 10;
		END_IF

	40:
		Initialize := TRUE;
END_CASE
END_METHOD

PROPERTY RcpProcess : REFERENCE TO ST_ProcessRecipe
GET
RcpProcess REF= _RcpProcess;
END_GET
END_PROPERTY

PROPERTY StsProcess : REFERENCE TO ST_ProcessStatus
GET
StsProcess REF= _StsProcess;
END_GET
END_PROPERTY

END_FUNCTION_BLOCK

// ---- Machine/02_EquipmentModules/03_Outfeed/EM_OutfeedModule.TcPOU
FUNCTION_BLOCK EM_OutfeedModule EXTENDS CommonModule IMPLEMENTS I_OutfeedModule
VAR
	//Components
	Axis : FB_Component_BasicAxis;

	//
	_CmdOutfeed : ST_OutfeedCommand;
	_StsOutfeed : ST_OutfeedStatus;
	_CfgOutfeed : ST_OutfeedConfig;
	_RcpOutfeed : ST_OutfeedRecipe;

	//Test Vars
	Homed : BOOL;
END_VAR

PROPERTY CfgOutfeed : REFERENCE TO ST_OutfeedConfig
GET
CfgOutfeed REF= _CfgOutfeed;
END_GET
END_PROPERTY

PROPERTY CmdOutfeed : REFERENCE TO ST_OutfeedCommand
GET
CmdOutfeed REF= _CmdOutfeed;
END_GET
END_PROPERTY

METHOD PUBLIC CyclicLogic
IF NOT _InitComplete THEN
	_InitComplete := Initialize();
	RETURN;
END_IF

SUPER^.CyclicLogic();
END_METHOD

//! @summary This method contains code which will execute when this PackML module is in the <b>Execute</b> state
METHOD PROTECTED Execute
(*! <description> <b>The base implementation of this method is empty. User must override this method to provide functionality.</b>
<table> 
	<tr>
		<th> Previous State </th>
		<th> Transition In </th>
		<th> Transition Out </th>
		<th> Next State  </th> 
	</tr>
	<tr>
		<td> Starting<b>-or-</b>Unholding <b>-or-</b>Unsuspending</td>
		<td> State Complete<i>(Starting<b>-or-</b>Unholding<b>-or-</b>Unsuspending)</i></td> 
		<td> State Complete<b>-or-</b>Hold Command<b>-or-</b>Suspend Command</td>
		<td> Completing<b>-or-</b>Holding<b>-or-</b>Suspending</td>
	</tr>
</table>
This method is called as required by <c>StateControl()</c>
</description> 

*)
VAR
END_VAR
CASE _CurrentMode OF
	E_PMLCustomMode.Production:
		CASE DescendantSequenceState OF
			0:
				IF _StsOutfeed.ProductAtReady THEN
					DescendantSequenceState := DescendantSequenceState + 10;
				END_IF

			10:
				IF Axis.MoveVelocity(10.0, 0) THEN
					DescendantSequenceState := DescendantSequenceState + 10;
				END_IF

			20:
				IF Axis.Axis.Status.Moving THEN
					_StsOutfeed.ProductAtReady	:= FALSE;
					_StsOutfeed.ConveyorRunning := TRUE;
				END_IF

				IF _StsOutfeed.ProductRemoved THEN
					_CmdOutfeed.StopConveyor := FALSE;
					Axis.Stop();
					DescendantSequenceState := DescendantSequenceState + 10;
				END_IF

			30:
				IF Axis.Axis.Status.NotMoving THEN
					_StsOutfeed.ConveyorRunning := FALSE;
					DescendantSequenceState		:= 0;
				END_IF
		END_CASE

	E_PMLCustomMode.Home:
		CASE DescendantSequenceState OF
			0:
				IF _CmdCommon.Home AND NOT _StsCommon.Homed THEN
					_CmdCommon.Home := FALSE;
					Axis.Home();
					DescendantSequenceState := DescendantSequenceState + 10;
				END_IF

			10:
				IF Axis.Axis.Status.Homed THEN
					_StsCommon.Homed := TRUE;
				END_IF
		END_CASE
END_CASE

SUPER^.Execute();
END_METHOD

METHOD PROTECTED Initialize : BOOL
VAR
	i: UDINT;
END_VAR
Initialize := FALSE;
CASE DescendantSequenceState OF
	0: //Register Modules

		//Register Components
		RegisterComponent(Axis);

		//I_CommonModuleBase

		//I_CommonComponent
		ipComponents[1] := Axis;

		//Setup Config
		_LogModeChanges			:= FALSE;
		_LogStateChanges		:= FALSE;
		DescendantSequenceState := DescendantSequenceState + 10;

	10:
		// Copy Mode names
		FOR i := 1 TO 10 DO
			ModeNames[i] := F_UnitModeToString(UDINT_TO_DINT(i));
		END_FOR

		DescendantSequenceState := DescendantSequenceState + 10;

	20:
		//Initialize_Recipes();
		DescendantSequenceState := DescendantSequenceState + 10;

	30: // Call the Super 
		IF SUPER^.Initialize() THEN
			DescendantSequenceState := DescendantSequenceState + 10;
		END_IF

	40:
		Initialize := TRUE;
END_CASE
END_METHOD

PROPERTY RcpOutfeed : REFERENCE TO ST_OutfeedRecipe
GET
RcpOutfeed REF= _RcpOutfeed;
END_GET
END_PROPERTY

PROPERTY StsOutfeed : REFERENCE TO ST_OutfeedStatus
GET
StsOutfeed REF= _StsOutfeed;
END_GET
END_PROPERTY

END_FUNCTION_BLOCK

// ---- Machine/03_Components/FB_Component_StackLight.TcPOU
FUNCTION_BLOCK FB_Component_StackLight EXTENDS CommonComponent
VAR
	
	//Alarms
	StackLightAlarm : ARRAY[1..ALARM_COUNT] OF FB_TcAlarm;
END_VAR
VAR CONSTANT
	ALARM_COUNT : INT := 2;
END_VAR

//! @summary Initializes event function blocks using this components's name
METHOD PROTECTED CreateEvents

//! @description This method is called by <c>Initialize()</c> as required
// Add your event creation here
(*F_CreateAllEventsInClass(Alarms		:= StackLightAlarm,
						 ClassSize	:= SIZEOF(TC_EVENTS.FestoServo),
						 pInitEvent := ADR(TC_EVENTS.FestoServo.InitReferenceEvent),
						 Prefix		:= _Name);*)

// Super call to base
SUPER^.CreateEvents();
END_METHOD

//! @summary This method serves as the entry point for all underlying FB logic
METHOD PUBLIC CyclicLogic

//! @description This method should be called cyclically by descendant function blocks by invoking <c>SUPER^.CyclicLogic()</c>.  Alternatively, the contents of this method could be reimplemented entirely in which case a call to this method would not be necessary.
SUPER^.CyclicLogic();

(* Update alarm severity from this component *)
_CurrentAlarmSeverity := F_GetMaxSeverityRaised(Alarms := StackLightAlarm, CurrentSeverity := _CurrentAlarmSeverity);
END_METHOD

//! Provides basic error detection and event handling for this component
METHOD PROTECTED Monitoring

(*! @descriptionThis method is called cyclically by <c>CyclicLogic()</c>*)
VAR
	i: INT;
END_VAR
IF _Error AND NOT StackLightAlarm[2].bRaised THEN
	RaiseAlarm2Args(StackLightAlarm[2], CONCAT('Error ID: ', TO_STRING(_ErrorID)), '');
END_IF

_Busy	 := _Busy;
_Error	 := _CurrentAlarmSeverity >= TcEventSeverity.Error;
_ErrorID := _ErrorID;
SUPER^.Monitoring();
END_METHOD

END_FUNCTION_BLOCK

// ---- POUs/Common/Component/CommonComponent.TcPOU
FUNCTION_BLOCK CommonComponent EXTENDS FB_ComponentBase
VAR
	ipCommonComponents : ARRAY[1..Parameters_PackML_Base.MAX_NO_OF_COMPONENTS] OF I_CommonComponent;
END_VAR

METHOD RaiseAlarm2Args
VAR_IN_OUT
    Alarm : FB_TcAlarm; //Alarm to be raised
END_VAR

VAR_INPUT
    String_1 : STRING; //First String Parameter (The Name of this component will be applied first automatically)
    String_2 : STRING; //Second String Parameter
END_VAR
F_RaiseAlarmWithStringParameters(Alarm    := Alarm,
                                 String_1 := Name,
                                 String_2 := String_1,
                                 String_3 := String_2);
END_METHOD

END_FUNCTION_BLOCK

// ---- Machine/03_Components/FB_Component_TwinSAFE_Monitor.TcPOU
FUNCTION_BLOCK FB_Component_TwinSAFE_Monitor EXTENDS CommonComponent
VAR
	//Alarms
	TwinSAFE_Alarms : ARRAY[1..ALARM_COUNT] OF FB_TcAlarm;
END_VAR

VAR CONSTANT
	ALARM_COUNT : INT := 2;
END_VAR

//! @summary Initializes event function blocks using this components's name
METHOD PROTECTED CreateEvents

//! @description This method is called by <c>Initialize()</c> as required
// Add your event creation here

(*F_CreateAllEventsInClass(Alarms		:= StackLightAlarm,
						 ClassSize	:= SIZEOF(TC_EVENTS.FestoServo),
						 pInitEvent := ADR(TC_EVENTS.FestoServo.InitReferenceEvent),
						 Prefix		:= _Name);*)

// Super call to base
SUPER^.CreateEvents();
END_METHOD

//! @summary This method serves as the entry point for all underlying FB logic
METHOD PUBLIC CyclicLogic

//! @description This method should be called cyclically by descendant function blocks by invoking <c>SUPER^.CyclicLogic()</c>.  Alternatively, the contents of this method could be reimplemented entirely in which case a call to this method would not be necessary.
SUPER^.CyclicLogic();

(* Update alarm severity from this component *)
_CurrentAlarmSeverity := F_GetMaxSeverityRaised(Alarms := TwinSAFE_Alarms, CurrentSeverity := _CurrentAlarmSeverity);
END_METHOD

//! Provides basic error detection and event handling for this component
METHOD PROTECTED Monitoring

(*! @descriptionThis method is called cyclically by <c>CyclicLogic()</c>*)
VAR
	i: INT;
END_VAR
IF _Error AND NOT TwinSAFE_Alarms[2].bRaised THEN
	RaiseAlarm2Args(TwinSAFE_Alarms[2], CONCAT('Error ID: ', TO_STRING(_ErrorID)), '');
END_IF

_Busy	 := _Busy;
_Error	 := _CurrentAlarmSeverity >= TcEventSeverity.Error;
_ErrorID := _ErrorID;
SUPER^.Monitoring();
END_METHOD

END_FUNCTION_BLOCK
